// TIA Portal V20 export
FUNCTION_BLOCK "FSFB_Main_Safety_RTG1"   // FB1, F_LAD
   VAR
      AllStopZone1 { ExternalAccessible := 'False'; ExternalVisible := 'False'; ExternalWritable := 'False'} : Bool;
      AllStopZone2 : Bool;
      Reset : Bool;
      Pair1 : ESTOP1;
      Pair2 : ESTOP1;
      Pair3 : ESTOP1;
      Pair4 : ESTOP1;
      Pair5 : ESTOP1;
      Pair6 : ESTOP1;
      Pair7 : ESTOP1;
      Pair8 : ESTOP1;
      Pair9 : ESTOP1;
      Pair10 : ESTOP1;
      ACK_GL : ACK_GL;
      ResetDelayTimer_Pair1 : TOF;
      ResetDelayTimer_Pair2 : TOF;
      ResetDelayTimer_Pair3 : TOF;
      ResetDelayTimer_Pair4 : TOF;
      ResetDelayTimer_Pair5 : TOF;
      ResetDelayTimer_Pair6 : TOF;
      ResetDelayTimer_Pair7 : TOF;
      ResetDelayTimer_Pair8 : TOF;
      ResetDelayTimer_Pair9 : TOF;
      ResetDelayTimer_Pair10 : TOF;
      mem_Pair1 : Bool;
      mem_Pair2 : Bool;
      mem_Pair3 : Bool;
      mem_Pair4 : Bool;
      mem_Pair5 : Bool;
      mem_Pair6 : Bool;
      mem_Pair7 : Bool;
      mem_Pair8 : Bool;
      mem_Pair9 : Bool;
      mem_Pair10 : Bool;
   END_VAR
   VAR_TEMP   // added for the SCL form of the ladder/FBD networks
      _w1 : Bool;
   END_VAR
BEGIN

REGION Network 1
   // Zone1
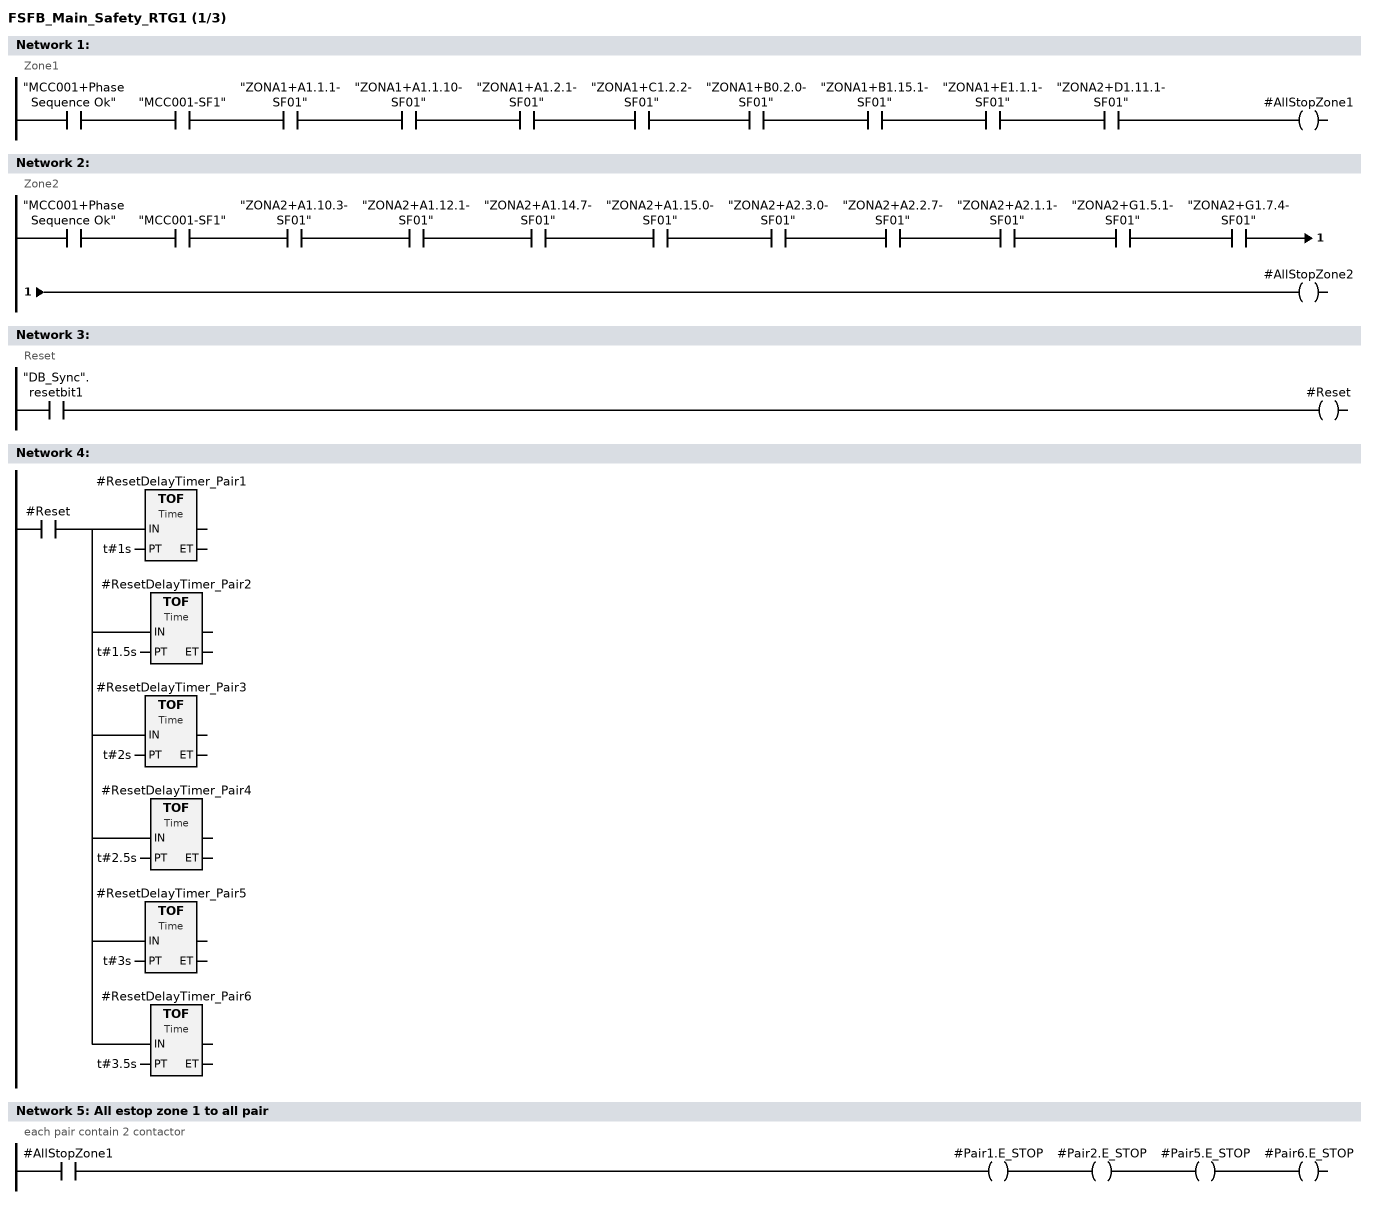
   RUNG wire#powerrail
      Contact( "MCC001+Phase Sequence Ok" )
      Contact( "MCC001-SF1" )
      Contact( "ZONA1+A1.1.1-SF01" )
      Contact( "ZONA1+A1.1.10-SF01" )
      Contact( "ZONA1+A1.2.1-SF01" )
      Contact( "ZONA1+C1.2.2-SF01" )
      Contact( "ZONA1+B0.2.0-SF01" )
      Contact( "ZONA1+B1.15.1-SF01" )
      Contact( "ZONA1+E1.1.1-SF01" )
      Contact( "ZONA2+D1.11.1-SF01" )
      Coil( #AllStopZone1 )
   END_RUNG
   // the same network as SCL:
   #AllStopZone1 := "MCC001+Phase Sequence Ok" AND "MCC001-SF1" AND "ZONA1+A1.1.1-SF01" AND "ZONA1+A1.1.10-SF01" AND "ZONA1+A1.2.1-SF01" AND "ZONA1+C1.2.2-SF01" AND "ZONA1+B0.2.0-SF01" AND "ZONA1+B1.15.1-SF01" AND "ZONA1+E1.1.1-SF01" AND "ZONA2+D1.11.1-SF01";
END_REGION

REGION Network 2
   // Zone2
   RUNG wire#powerrail
      Contact( "MCC001+Phase Sequence Ok" )
      Contact( "MCC001-SF1" )
      Contact( "ZONA2+A1.10.3-SF01" )
      Contact( "ZONA2+A1.12.1-SF01" )
      Contact( "ZONA2+A1.14.7-SF01" )
      Contact( "ZONA2+A1.15.0-SF01" )
      Contact( "ZONA2+A2.3.0-SF01" )
      Contact( "ZONA2+A2.2.7-SF01" )
      Contact( "ZONA2+A2.1.1-SF01" )
      Contact( "ZONA2+G1.5.1-SF01" )
      Contact( "ZONA2+G1.7.4-SF01" )
      Coil( #AllStopZone2 )
   END_RUNG
   // the same network as SCL:
   #AllStopZone2 := "MCC001+Phase Sequence Ok" AND "MCC001-SF1" AND "ZONA2+A1.10.3-SF01" AND "ZONA2+A1.12.1-SF01" AND "ZONA2+A1.14.7-SF01" AND "ZONA2+A1.15.0-SF01" AND "ZONA2+A2.3.0-SF01" AND "ZONA2+A2.2.7-SF01" AND "ZONA2+A2.1.1-SF01" AND "ZONA2+G1.5.1-SF01" AND "ZONA2+G1.7.4-SF01";
END_REGION

REGION Network 3
   // Reset
   RUNG wire#powerrail
      Contact( "DB_Sync".resetbit1 )
      Coil( #Reset )
   END_RUNG
   // the same network as SCL:
   #Reset := "DB_Sync".resetbit1;
END_REGION

REGION Network 4
   RUNG wire#powerrail
      Contact( #Reset )
      wire#w1
      { S7_Templates := "[time_type := Time, codedbool_type := DInt]" } #ResetDelayTimer_Pair1.TOF(pt := t#1s, et =>)
   END_RUNG
   RUNG wire#w1
      { S7_Templates := "[time_type := Time, codedbool_type := DInt]" } #ResetDelayTimer_Pair2.TOF(pt := t#1.5s, et =>)
   END_RUNG
   RUNG wire#w1
      { S7_Templates := "[time_type := Time, codedbool_type := DInt]" } #ResetDelayTimer_Pair3.TOF(pt := t#2s, et =>)
   END_RUNG
   RUNG wire#w1
      { S7_Templates := "[time_type := Time, codedbool_type := DInt]" } #ResetDelayTimer_Pair4.TOF(pt := t#2.5s, et =>)
   END_RUNG
   RUNG wire#w1
      { S7_Templates := "[time_type := Time, codedbool_type := DInt]" } #ResetDelayTimer_Pair5.TOF(pt := t#3s, et =>)
   END_RUNG
   RUNG wire#w1
      { S7_Templates := "[time_type := Time, codedbool_type := DInt]" } #ResetDelayTimer_Pair6.TOF(pt := t#3.5s, et =>)
   END_RUNG
   // the same network as SCL:
   #ResetDelayTimer_Pair1.TOF(IN := #Reset, PT := t#1s);
   #ResetDelayTimer_Pair2.TOF(IN := #Reset, PT := t#1.5s);
   #ResetDelayTimer_Pair3.TOF(IN := #Reset, PT := t#2s);
   #ResetDelayTimer_Pair4.TOF(IN := #Reset, PT := t#2.5s);
   #ResetDelayTimer_Pair5.TOF(IN := #Reset, PT := t#3s);
   #ResetDelayTimer_Pair6.TOF(IN := #Reset, PT := t#3.5s);
END_REGION

REGION Network 5: All estop zone 1 to all pair
   // each pair contain 2 contactor
   RUNG wire#powerrail
      Contact( #AllStopZone1 )
      Coil( #Pair1.E_STOP )
      Coil( #Pair2.E_STOP )
      Coil( #Pair5.E_STOP )
      Coil( #Pair6.E_STOP )
   END_RUNG
   // the same network as SCL:
   #Pair1.E_STOP := #AllStopZone1;
   #Pair2.E_STOP := #AllStopZone1;
   #Pair5.E_STOP := #AllStopZone1;
   #Pair6.E_STOP := #AllStopZone1;
END_REGION

REGION Network 6: All estop zone 2 to all pair
   // each pair contain 2 contactor
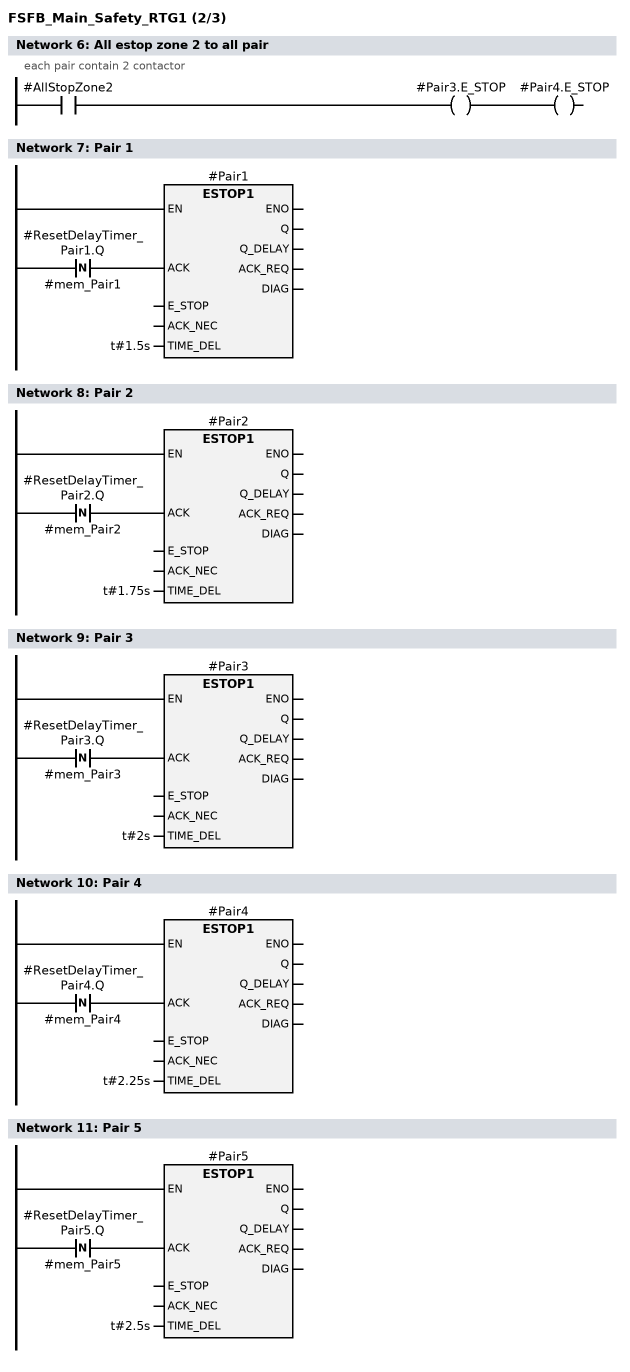
   RUNG wire#powerrail
      Contact( #AllStopZone2 )
      Coil( #Pair3.E_STOP )
      Coil( #Pair4.E_STOP )
   END_RUNG
   // the same network as SCL:
   #Pair3.E_STOP := #AllStopZone2;
   #Pair4.E_STOP := #AllStopZone2;
END_REGION

REGION Network 7: Pair 1
   RUNG wire#powerrail
      #Pair1.ESTOP1(ACK := wire#w1, E_STOP :=, ACK_NEC :=, TIME_DEL := t#1.5s, Q =>, Q_DELAY =>, ACK_REQ =>, DIAG =>)
   END_RUNG
   RUNG wire#powerrail
      N_Contact(operand := #ResetDelayTimer_Pair1.Q, bit := #mem_Pair1)
   END_RUNG wire#w1
   // the same network as SCL:
   #_w1 := NOT #ResetDelayTimer_Pair1.Q AND #mem_Pair1;   // falling edge of #ResetDelayTimer_Pair1.Q
   #mem_Pair1 := #ResetDelayTimer_Pair1.Q;
   #Pair1(ACK := #_w1, TIME_DEL := t#1.5s);   // ESTOP1
END_REGION

REGION Network 8: Pair 2
   RUNG wire#powerrail
      #Pair2.ESTOP1(ACK := wire#w1, E_STOP :=, ACK_NEC :=, TIME_DEL := t#1.75s, Q =>, Q_DELAY =>, ACK_REQ =>, DIAG =>)
   END_RUNG
   RUNG wire#powerrail
      N_Contact(operand := #ResetDelayTimer_Pair2.Q, bit := #mem_Pair2)
   END_RUNG wire#w1
   // the same network as SCL:
   #_w1 := NOT #ResetDelayTimer_Pair2.Q AND #mem_Pair2;   // falling edge of #ResetDelayTimer_Pair2.Q
   #mem_Pair2 := #ResetDelayTimer_Pair2.Q;
   #Pair2(ACK := #_w1, TIME_DEL := t#1.75s);   // ESTOP1
END_REGION

REGION Network 9: Pair 3
   RUNG wire#powerrail
      #Pair3.ESTOP1(ACK := wire#w1, E_STOP :=, ACK_NEC :=, TIME_DEL := t#2s, Q =>, Q_DELAY =>, ACK_REQ =>, DIAG =>)
   END_RUNG
   RUNG wire#powerrail
      N_Contact(operand := #ResetDelayTimer_Pair3.Q, bit := #mem_Pair3)
   END_RUNG wire#w1
   // the same network as SCL:
   #_w1 := NOT #ResetDelayTimer_Pair3.Q AND #mem_Pair3;   // falling edge of #ResetDelayTimer_Pair3.Q
   #mem_Pair3 := #ResetDelayTimer_Pair3.Q;
   #Pair3(ACK := #_w1, TIME_DEL := t#2s);   // ESTOP1
END_REGION

REGION Network 10: Pair 4
   RUNG wire#powerrail
      #Pair4.ESTOP1(ACK := wire#w1, E_STOP :=, ACK_NEC :=, TIME_DEL := t#2.25s, Q =>, Q_DELAY =>, ACK_REQ =>, DIAG =>)
   END_RUNG
   RUNG wire#powerrail
      N_Contact(operand := #ResetDelayTimer_Pair4.Q, bit := #mem_Pair4)
   END_RUNG wire#w1
   // the same network as SCL:
   #_w1 := NOT #ResetDelayTimer_Pair4.Q AND #mem_Pair4;   // falling edge of #ResetDelayTimer_Pair4.Q
   #mem_Pair4 := #ResetDelayTimer_Pair4.Q;
   #Pair4(ACK := #_w1, TIME_DEL := t#2.25s);   // ESTOP1
END_REGION

REGION Network 11: Pair 5
   RUNG wire#powerrail
      #Pair5.ESTOP1(ACK := wire#w1, E_STOP :=, ACK_NEC :=, TIME_DEL := t#2.5s, Q =>, Q_DELAY =>, ACK_REQ =>, DIAG =>)
   END_RUNG
   RUNG wire#powerrail
      N_Contact(operand := #ResetDelayTimer_Pair5.Q, bit := #mem_Pair5)
   END_RUNG wire#w1
   // the same network as SCL:
   #_w1 := NOT #ResetDelayTimer_Pair5.Q AND #mem_Pair5;   // falling edge of #ResetDelayTimer_Pair5.Q
   #mem_Pair5 := #ResetDelayTimer_Pair5.Q;
   #Pair5(ACK := #_w1, TIME_DEL := t#2.5s);   // ESTOP1
END_REGION

REGION Network 12: Pair 6
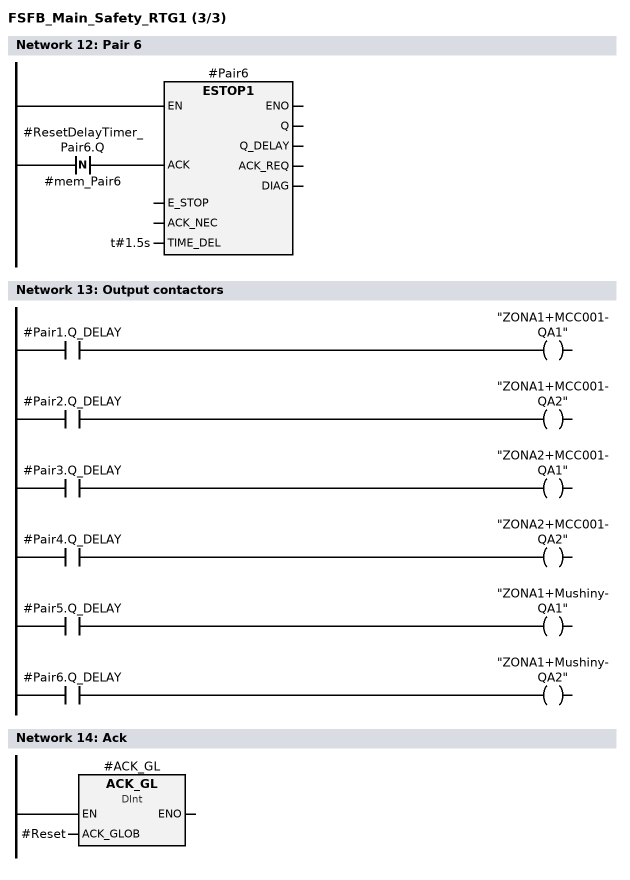
   RUNG wire#powerrail
      #Pair6.ESTOP1(ACK := wire#w1, E_STOP :=, ACK_NEC :=, TIME_DEL := t#1.5s, Q =>, Q_DELAY =>, ACK_REQ =>, DIAG =>)
   END_RUNG
   RUNG wire#powerrail
      N_Contact(operand := #ResetDelayTimer_Pair6.Q, bit := #mem_Pair6)
   END_RUNG wire#w1
   // the same network as SCL:
   #_w1 := NOT #ResetDelayTimer_Pair6.Q AND #mem_Pair6;   // falling edge of #ResetDelayTimer_Pair6.Q
   #mem_Pair6 := #ResetDelayTimer_Pair6.Q;
   #Pair6(ACK := #_w1, TIME_DEL := t#1.5s);   // ESTOP1
END_REGION

REGION Network 13: Output contactors
   RUNG wire#powerrail
      Contact( #Pair1.Q_DELAY )
      Coil( "ZONA1+MCC001-QA1" )
   END_RUNG
   RUNG wire#powerrail
      Contact( #Pair2.Q_DELAY )
      Coil( "ZONA1+MCC001-QA2" )
   END_RUNG
   RUNG wire#powerrail
      Contact( #Pair3.Q_DELAY )
      Coil( "ZONA2+MCC001-QA1" )
   END_RUNG
   RUNG wire#powerrail
      Contact( #Pair4.Q_DELAY )
      Coil( "ZONA2+MCC001-QA2" )
   END_RUNG
   RUNG wire#powerrail
      Contact( #Pair5.Q_DELAY )
      Coil( "ZONA1+Mushiny-QA1" )
   END_RUNG
   RUNG wire#powerrail
      Contact( #Pair6.Q_DELAY )
      Coil( "ZONA1+Mushiny-QA2" )
   END_RUNG
   // the same network as SCL:
   "ZONA1+MCC001-QA1" := #Pair1.Q_DELAY;
   "ZONA1+MCC001-QA2" := #Pair2.Q_DELAY;
   "ZONA2+MCC001-QA1" := #Pair3.Q_DELAY;
   "ZONA2+MCC001-QA2" := #Pair4.Q_DELAY;
   "ZONA1+Mushiny-QA1" := #Pair5.Q_DELAY;
   "ZONA1+Mushiny-QA2" := #Pair6.Q_DELAY;
END_REGION

REGION Network 14: Ack
   RUNG wire#powerrail
      { S7_Templates := "codedbool_type := DInt" } #ACK_GL.ACK_GL(ACK_GLOB := #Reset)
   END_RUNG
   // the same network as SCL:
   #ACK_GL(ACK_GLOB := #Reset);   // ACK_GL
END_REGION
END_FUNCTION_BLOCK
